{attribute addProperty BoxType "EL6201-0000-0017"}
{attribute addProperty Id "Slave_9A_DI0BIT10.12565Slave_9A_DI1BIT10.12566Slave_9A_DI2BIT10.12567Slave_9A_DI3BIT10.12568Slave_9B_DI0BIT10.12569Slave_9B_DI1BIT10.12570Slave_9B_DI2BIT10.12571Slave_9B_DI3BIT10.12572"}
{attribute addProperty CRC "2031410654"}
{attribute addProperty SizeInBites "8"}
{attribute addProperty SizeInBytes "1"}
TYPE Slave_9_Inputs_7914DDDE :
STRUCT
	{attribute addProperty Name "Slave_9A_DI0"}
	Slave_9A_DI0 : BIT;
	{attribute addProperty Name "Slave_9A_DI1"}
	Slave_9A_DI1 : BIT;
	{attribute addProperty Name "Slave_9A_DI2"}
	Slave_9A_DI2 : BIT;
	{attribute addProperty Name "Slave_9A_DI3"}
	Slave_9A_DI3 : BIT;
	{attribute addProperty Name "Slave_9B_DI0"}
	Slave_9B_DI0 : BIT;
	{attribute addProperty Name "Slave_9B_DI1"}
	Slave_9B_DI1 : BIT;
	{attribute addProperty Name "Slave_9B_DI2"}
	Slave_9B_DI2 : BIT;
	{attribute addProperty Name "Slave_9B_DI3"}
	Slave_9B_DI3 : BIT;
END_STRUCT
END_TYPE

(* stored: Version 1.2.0.0, ProductVersion 3.1.4024.9
   DUT Slave_9_Inputs_7914DDDE: Id {edf71221-cc66-44c6-8c28-78f06a88aa86} *)
